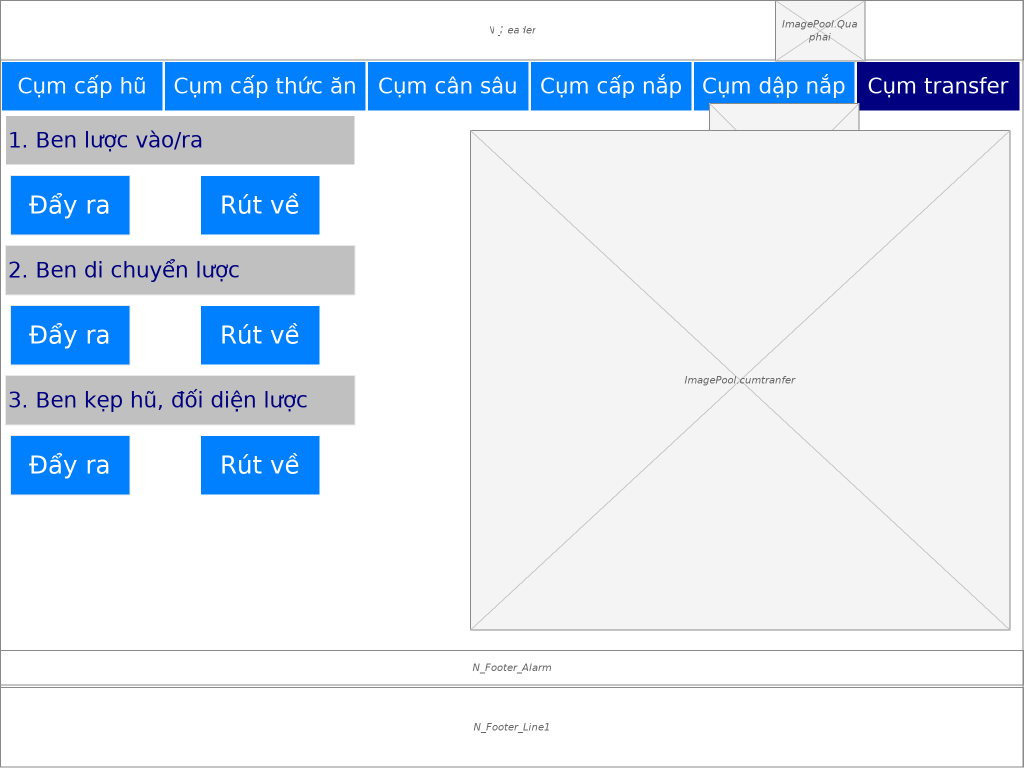
VISUALIZATION N_Tranfer1  // 1024x768
    Rectangle (10,305 120x60), "Đẩy ra", colour toggle: PR_Line01.bCylinder_Move_Comb_Extend, input disabled if: Not PR_Line01.bCheck
        OnMouseDown: execute {
            PR_Line01.bCylinder_Move_Comb_Extend := TRUE;
            PR_Line01.bCylinder_Move_Comb_Retract := FALSE;
            PR_Line01.bxa := FALSE;
        }
    Rectangle (200,175 120x60), "Rút về", colour toggle: PR_Line01.bCylinder_Comb_Retract
        OnMouseDown: execute {
            PR_Line01.bCylinder_Comb_Retract := TRUE;
            PR_Line01.bCylinder_Comb_Extend := FALSE;
            PR_Line01.bxa := FALSE;
        }
    Rectangle (200,305 120x60), "Rút về", colour toggle: PR_Line01.bCylinder_Move_Comb_Retract, input disabled if: Not PR_Line01.bCheck
        OnMouseDown: execute {
            PR_Line01.bCylinder_Move_Comb_Retract := TRUE;
            PR_Line01.bCylinder_Move_Comb_Extend := FALSE;
            PR_Line01.bxa := FALSE;
        }
    Frame (0,687 1024x80)
        shows N_Footer_Line1()
    Frame (0,0 1024x60)
        shows N_Header()
    Textfield (353,5 400x50), "MÀN HÌNH CHẠY TAY LINE 1"
    Rectangle (5,115 350x50), "1. Ben lược vào/ra"
    Rectangle (10,175 120x60), "Đẩy ra", colour toggle: PR_Line01.bCylinder_Comb_Extend, input disabled if: Not PR_Line01.bCheck
        OnMouseDown: execute {
            PR_Line01.bCylinder_Comb_Extend := TRUE;
            PR_Line01.bCylinder_Comb_Retract := FALSE;
            PR_Line01.bxa := FALSE;
        }
    Rectangle (5,245 350x50), "2. Ben di chuyển lược"
    Rectangle (1,61 162x50), "Cụm cấp hũ"
        OnMouseClick: change screen: N_JarSupply1
    Rectangle (164,61 202x50), "Cụm cấp thức ăn"
        OnMouseClick: change screen: N_FoodSupply1
    Rectangle (367,61 162x50), "Cụm cân sâu"
        OnMouseClick: change screen: N_WormWeight1
    Rectangle (530,61 162x50), "Cụm cấp nắp"
        OnMouseClick: change screen: N_LidSupply1
    Rectangle (693,61 162x50), "Cụm dập nắp"
        OnMouseClick: change screen: N_LidPressing1
    Rectangle (856,61 164x50), "Cụm transfer"
        OnMouseClick: change screen: N_Tranfer1
    Rectangle (5,375 350x50), "3. Ben kẹp hũ, đối diện lược"
    Rectangle (200,435 120x60), "Rút về", text variable: GVL_OF_VU.fFreqOutputConveyor, colour toggle: PR_Line01.bCylinder_Clip_Retract
        OnMouseDown: execute {
            PR_Line01.bCylinder_Clip_Retract := TRUE;
            PR_Line01.bCylinder_Clip_Extend := FALSE;
            PR_Line01.bxa := FALSE;
        }
    Rectangle (10,435 120x60), "Đẩy ra", colour toggle: PR_Line01.bCylinder_Clip_Extend
        OnMouseDown: execute {
            PR_Line01.bCylinder_Clip_Extend := TRUE;
            PR_Line01.bCylinder_Clip_Retract := FALSE;
            PR_Line01.bxa := FALSE;
        }
    Image (709,103 150x150)
    Image (775,0 90x61), image: ImagePool.Qua phai
        OnMouseClick: change screen: N_Tranfer2
        OnMouseClick: execute { MAIN_LINE2.bModeManual := TRUE; MAIN_LINE2.bModeAuto := FALSE; }
    Image (470,130 540x500), image: ImagePool.cumtranfer
    Frame (0,650 1024x35)
        shows N_Footer_Alarm()
END_VISUALIZATION

(* stored: Version 1.1.0.1, ProductVersion 3.1.4024.12
   Visu N_Tranfer1: Id {7b0d379c-c4f0-4d05-aa8f-bb4b7442d513} *)
